FUNCTION_BLOCK E_MERGE_2 (* Merge (OR) of two input events *)
  (* Standard: 61499-1 Annex A; Function: Output EO is triggered when either EI1 or EI2 is received; Description: Copyright (c) 2017 fortiss GmbH This program and the accompanying materials are made available under the terms of the Eclipse Public License 2.0 which is available at https://www.eclipse.org/legal/epl-2.0/ SPDX-License-Identifier: EPL-2.0 *)
  (* Version 1.0, 2017, Alois Zoitl, fortiss GmbH, initial API and implementation and/or initial documentation *)
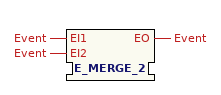
  EVENT_INPUT
    EI1; (* First input event *)
    EI2; (* Second input event *)
  END_EVENT
  EVENT_OUTPUT
    EO; (* Output Event *)
  END_EVENT
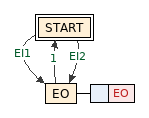
  EC_STATES
    START; (* Initial State *)
    EO : -> EO; (* Issue EO Event *)
  END_STATES
  EC_TRANSITIONS
    EO TO START := 1;
    START TO EO := EI1;
    START TO EO := EI2;
  END_TRANSITIONS
END_FUNCTION_BLOCK
